// TIA Portal V20 export
TYPE "Temporizadores_flujos_mesa"
   STRUCT
      MAUX_INICIO_REGISTRO : Bool;
      MAUX_FIN_REGISTRO : Bool;
      NUM_REGISTRO_ACTUAL { ExternalAccessible := 'False'; ExternalVisible := 'False'; ExternalWritable := 'False'} : Int;
      TMP_Etapas_Carga_E0 { S7_SetPoint := 'True'} : TONR_TIME;
      TMP_Etapas_Carga_E1 { S7_SetPoint := 'True'} : TONR_TIME;
      TMP_Etapas_Carga_E2 { S7_SetPoint := 'True'} : TONR_TIME;
      TMP_Etapas_Carga_E3 { S7_SetPoint := 'True'} : TONR_TIME;
      TMP_Etapas_Carga_E4 { S7_SetPoint := 'True'} : TONR_TIME;
      TMP_Etapas_Descarga_S0 { S7_SetPoint := 'True'} : TONR_TIME;
      TMP_Etapas_Descarga_S1 { S7_SetPoint := 'True'} : TONR_TIME;
      TMP_Etapas_Descarga_S2 { S7_SetPoint := 'True'} : TONR_TIME;
      TMP_Etapas_Descarga_S3 { S7_SetPoint := 'True'} : TONR_TIME;
      TMP_Etapas_Descarga_S4 { S7_SetPoint := 'True'} : TONR_TIME;
      TMP_Etapa_Cargada { S7_SetPoint := 'True'} : TONR_TIME;
      TMP_AvanceRetroceso_Cadenas { S7_SetPoint := 'True'} : TONR_TIME;
      TMP_AvanceRetroceso_Rodillos { S7_SetPoint := 'True'} : TONR_TIME;
      TMP_Giro { S7_SetPoint := 'True'} : TONR_TIME;
      TMP_Subir_Transfer { S7_SetPoint := 'True'} : TONR_TIME;
      TMP_Bajar_Transfer { S7_SetPoint := 'True'} : TONR_TIME;
   END_STRUCT;
END_TYPE
